// LS Electric XG5000 project: 컨베이어_테스트
// PLC NewPLC

PROGRAM HMI_PLC_입력중계 (task: 스캔 프로그램)

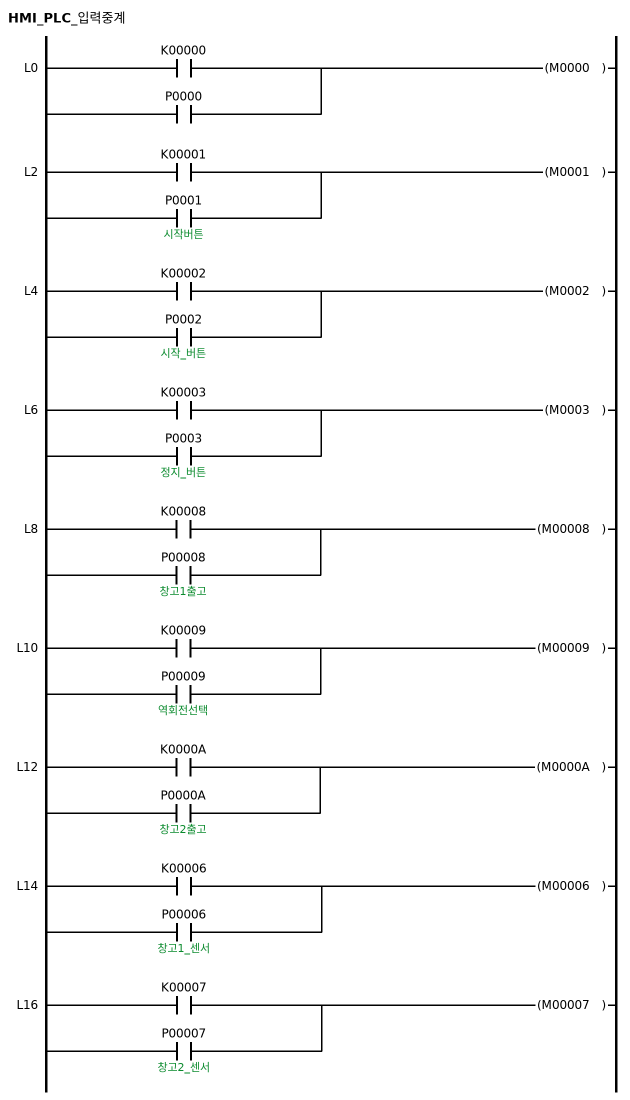
; L0
LOAD      K00000
OR        P0000
OUT       M0000
; L2
LOAD      K00001
OR        P0001	// 시작버튼
OUT       M0001
; L4
LOAD      K00002
OR        P0002	// 시작_버튼
OUT       M0002
; L6
LOAD      K00003
OR        P0003	// 정지_버튼
OUT       M0003
; L8
LOAD      K00008
OR        P00008	// 창고1출고
OUT       M00008
; L10
LOAD      K00009
OR        P00009	// 역회전선택
OUT       M00009
; L12
LOAD      K0000A
OR        P0000A	// 창고2출고
OUT       M0000A
; L14
LOAD      K00006
OR        P00006	// 창고1_센서
OUT       M00006
; L16
LOAD      K00007
OR        P00007	// 창고2_센서
OUT       M00007

PROGRAM 컨베이어_시스템 (task: 스캔 프로그램)

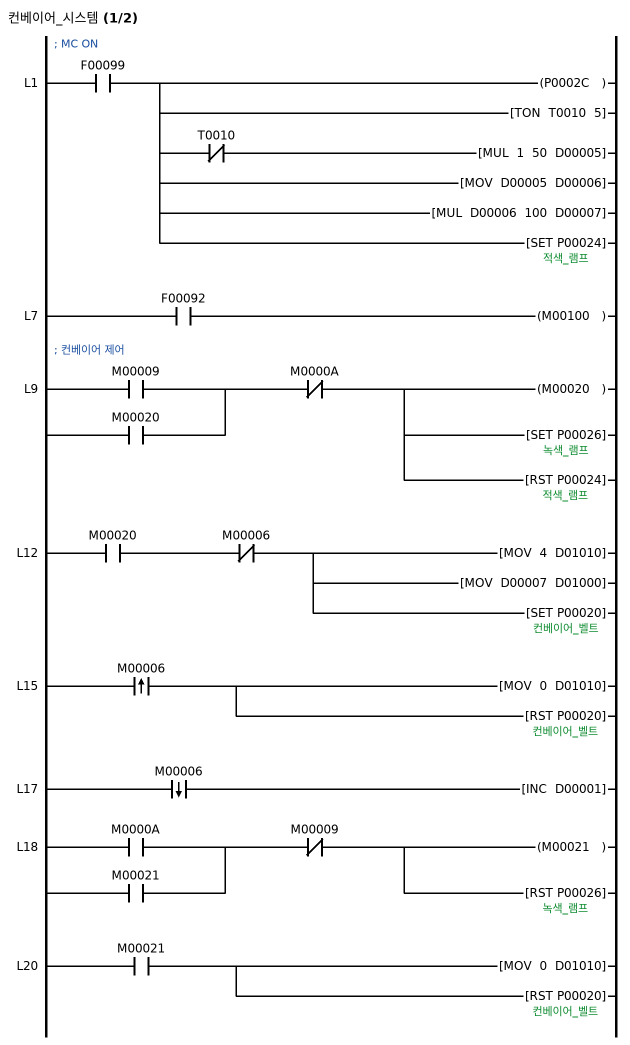
// MC ON
; L1
LOAD      F00099
OUT       P0002C
TON       T0010 5
MPUSH
AND NOT   T0010
MUL       1 50 D00005
MPOP
MOV       D00005 D00006
MUL       D00006 100 D00007
SET       P00024	// 적색_램프
; L7
LOAD      F00092
OUT       M00100
// 컨베이어 제어
; L9
LOAD      M00009
OR        M00020
AND NOT   M0000A
OUT       M00020
SET       P00026	// 녹색_램프
RST       P00024	// 적색_램프
; L12
LOAD      M00020
AND NOT   M00006
MOV       4 D01010
MOV       D00007 D01000
SET       P00020	// 컨베이어_벨트
; L15
LOADP     M00006
MOV       0 D01010
RST       P00020	// 컨베이어_벨트
; L17
LOADN     M00006
INC       D00001
; L18
LOAD      M0000A
OR        M00021
AND NOT   M00009
OUT       M00021
RST       P00026	// 녹색_램프
; L20
LOAD      M00021
MOV       0 D01010
RST       P00020	// 컨베이어_벨트

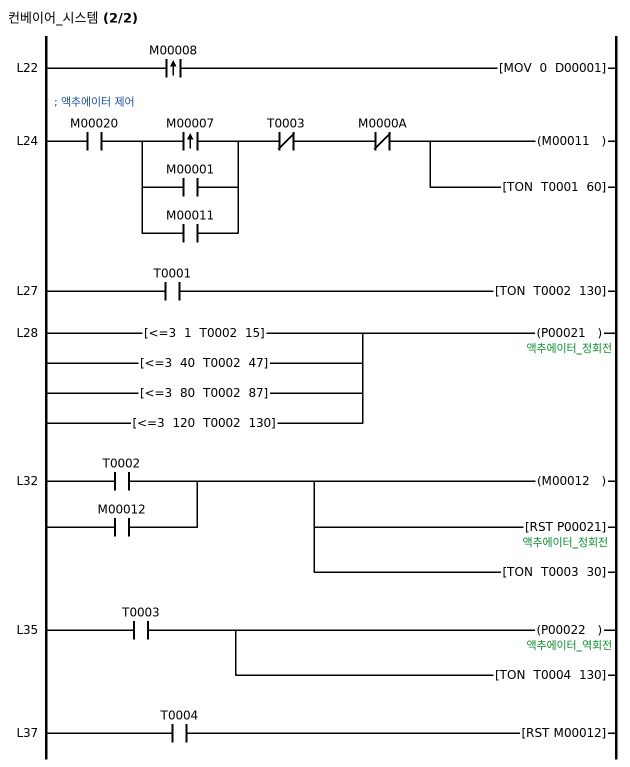
; L22
LOADP     M00008
MOV       0 D00001
// 액추에이터 제어
; L24
LOAD      M00020
LOADP     M00007
OR        M00001
OR        M00011
AND LOAD
AND NOT   T0003
AND NOT   M0000A
OUT       M00011
TON       T0001 60
; L27
LOAD      T0001
TON       T0002 130
; L28
LOAD<=3   1 T0002 15
OR<=3     40 T0002 47
OR<=3     80 T0002 87
OR<=3     120 T0002 130
OUT       P00021	// 액추에이터_정회전
; L32
LOAD      T0002
OR        M00012
OUT       M00012
RST       P00021	// 액추에이터_정회전
TON       T0003 30
; L35
LOAD      T0003
OUT       P00022	// 액추에이터_역회전
TON       T0004 130
; L37
LOAD      T0004
RST       M00012

VARIABLES AND COMMENTS (devices not used above)
P0000D	BIT	램프_1
P0000E	BIT	램프_2
P00025	BIT	신호기2_황색
P00029	BIT	신호기3_좌회전
P00023	BIT	신호등1_적색
P00027	BIT	신호등3_적색
P00028	BIT	신호등3_황색
P0000B	BIT	정지
P00004	BIT	창고1_출고
P00005	BIT	창고2_출고